Yaskawa INFORM job: TESTTCPKM.JBI

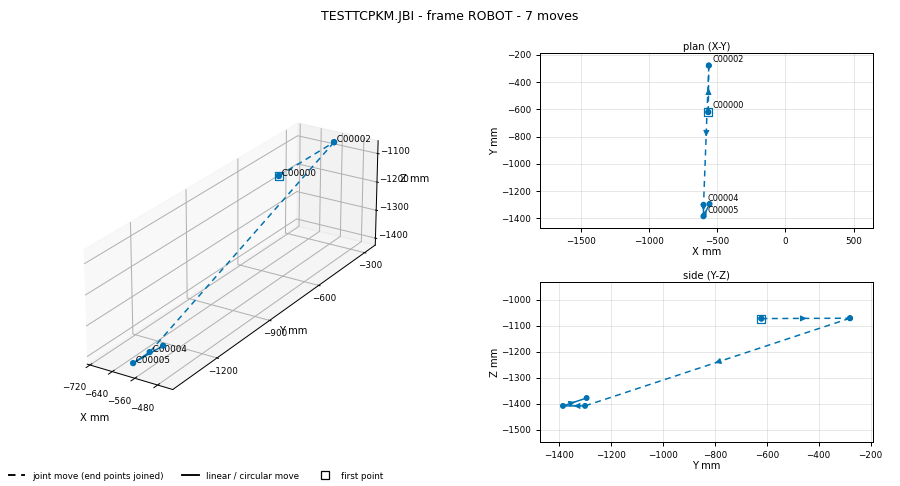
[picture p0: tool path of TESTTCPKM.JBI in frame ROBOT, 7 of 7 moves have a stored position in this frame; points joined in program order, loops and branches not executed]
/JOB
//NAME TESTTCPKM
//POS
///NPOS 7,7,7,0,0,0
///TOOL 0
///POSTYPE ROBOT
///RECTAN
///RCONF 0,0,0,0,1,0,0,0,0,0,0,0,0,0,0,0,0,0,0,0,0,0,0,0
C00000=-565.623,-620.809,-1072.434,67.8686,14.8572,-179.0143
C00001=-565.623,-620.809,-1072.434,67.8686,14.8572,-179.0143
///RCONF 0,0,0,0,0,0,0,0,0,0,0,0,0,0,0,0,0,0,0,0,0,0,0,0
C00002=-561.741,-279.159,-1071.117,-64.8250,5.1767,-48.0999
C00003=-561.741,-279.159,-1071.117,-64.8250,5.1767,-48.0999
C00004=-600.242,-1300.014,-1408.903,-46.0047,8.4003,-73.6799
C00005=-601.209,-1385.146,-1409.006,-46.0054,8.3991,-73.6804
C00006=-555.934,-1293.987,-1378.499,-46.0039,8.3996,-73.6811
BC00000=2467.273,352.367,802.962
BC00001=2467.273,352.367,802.962
BC00002=2467.273,9.811,801.315
BC00003=2467.273,9.811,801.315
BC00004=2481.977,2113.917,622.333
BC00005=2481.977,2113.917,622.333
BC00006=2481.977,2113.917,622.333
///POSTYPE PULSE
///PULSE
EC00000=-1,-1
EC00001=-1,-1
EC00002=-1,-1
EC00003=-1,-1
EC00004=-1,0
EC00005=-1,0
EC00006=-1,0
//INST
///DATE 2023/11/23 14:25
///ATTR SC,RW,RJ
////FRAME ROBOT
///GROUP1 RB1,BS1
///GROUP2 ST1
NOP
MOVJ C00000 BC00000 VJ=0.78  +MOVJ EC00000 VJ=0.78
MOVL C00001 BC00001 V=11.0  +MOVJ EC00001 VJ=0.78
MOVJ C00002 BC00002 VJ=0.78  +MOVJ EC00002 VJ=0.78
MOVL C00003 BC00003 V=11.0  +MOVJ EC00003 VJ=0.78
MOVJ C00004 BC00004 VJ=100.00  +MOVJ EC00004 VJ=100.00
MACRO1 MJ#(0) ARGF9
ARCON
MOVL C00005 BC00005 V=9.2  +MOVJ EC00005 VJ=100.00
ARCOF
MOVL C00006 BC00006 V=33.3  +MOVJ EC00006 VJ=100.00
PAUSE
END
